RoboDK station: PDE4431_CW2_Final_Station4.rdk

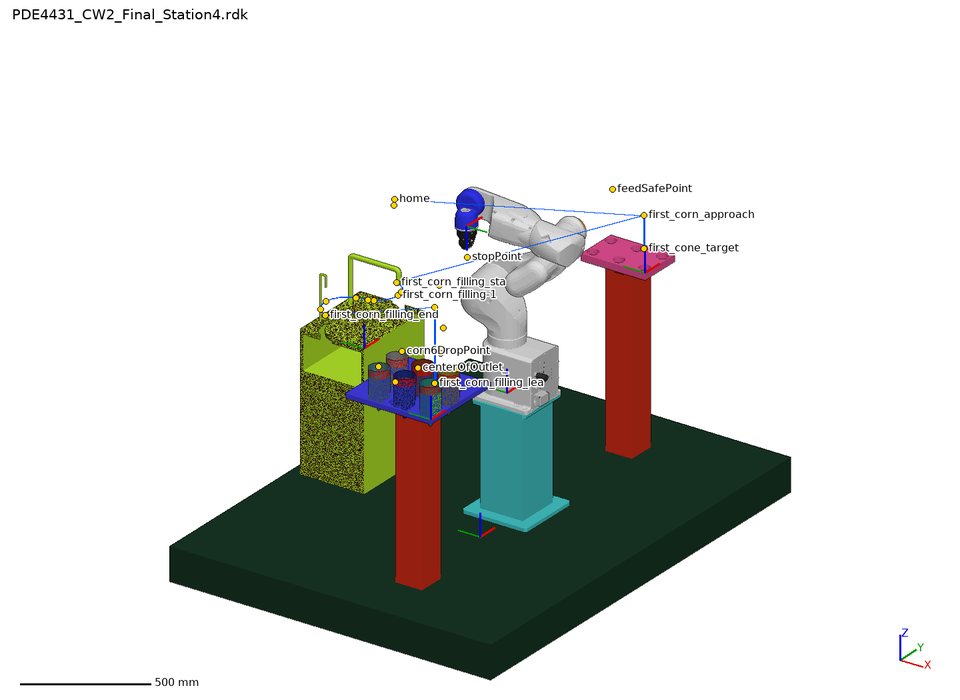
[picture v0: the station drawn from its stored meshes, robots at their saved joint values, targets as dots, program paths as lines]
Station PDE4431_CW2_Final_Station4 (saved by RoboDK 5.8.0). Poses are relative to the parent item; angles as X-Y-Z fixed-axis rotations.
  - frame world_frame at (0, 0, 10) mm, rotated rx 0 ry 0 rz 90 deg
    - object PDE4431_CW2_2024 at (0, 0, 0) mm, rotated rx 90 ry 0 rz 0 deg, size 2000 x 980 x 1500 mm, geometry from PDE4431_CW2_2024.STEP
    - object Pedestal_3 at (28, -150, 150) mm, rotated rx 90 ry 0 rz 0 deg, size 300 x 480 x 300 mm, geometry from Pedestal_3.STEP
    - frame Epson VT6 Base at (30, -105, 630) mm
      - robot Epson VT6: 6 axes, payload 6 kg, reach 920 mm, repeatability 0.1 mm, weight 40 kg
          modified DH rows (alpha deg, a mm, theta deg, d mm): 0, 0, 0, 412; -90, 100, -90, 0; 0, 420, 0, 0; -90, 0, 0, 400; 90, 0, 0, 0; -90, 0, 0, 80
          base shift (0, 0, 0) mm, rotated rx 0 ry 0 rz 90 deg
          joint limits [-170, -160, -51, -200, -125, -360] to [170, 65, 190, 200, 125, 360]; home [0, 0, 0, 0, 0, 0]; saved at [8.367, 49.246, -40.116, -0.033, -101.34, -10.833]
        - frame RobotiQ 2F-85 Gripper (Mechanism) Base at (0, 0, 0) mm, rotated rx 0 ry 0 rz 90 deg
          - robot RobotiQ 2F-85 Gripper (Mechanism) (model RobotiQ 2F85): 1 axes, payload 5 kg
              joint limits [0] to [85]; home [85]; saved at [60]
        - tool Tool 1, TCP at (0, 0, 130) mm
      - target gripper_open (Cartesian target) at (0, 683.92, 832) mm, rotated rx -90 ry 0 rz 0 deg; joints [85, 0, 0, 0, 0, 0] of RobotiQ 2F-85 Gripper (Mechanism)
      - target gripper_close (Cartesian target) at (0, 683.92, 832) mm, rotated rx -90 ry 0 rz 0 deg; joints [60, 0, 0, 0, 0, 0] of RobotiQ 2F-85 Gripper (Mechanism)
    - frame feed_frame at (600, -350, 980) mm
      - target home (Cartesian target) at (-608.8, 742.44, 350) mm, rotated rx 19.99 ry -88.06 rz -110.51 deg; joints [1.443, 8.858, -28.234, -5.378, 21.283, 5.738] of Epson VT6
      - target first_cone_target (Cartesian target) at (40.44, 31.41, 80) mm, rotated rx 9.95 ry -88.07 rz 169.53 deg; joints [-105.167, -26.118, -40.115, 15.72, 68.941, -5.939] of Epson VT6
      - target first_corn_approach (Cartesian target) at (40.44, 31.41, 220) mm, rotated rx 9.95 ry -88.07 rz 169.53 deg; joints [-123.826, -9.454, -31.705, 43.687, 52.628, -31.019] of Epson VT6
      - target first_corn_filling-1 (Cartesian target) at (-501.04, 802, -119.95) mm, rotated rx 9.87 ry -88.07 rz -104.39 deg; joints [-10.546, -59.86, -31.979, 6.038, 93.729, 0.524] of Epson VT6
      - target first_corn_filling_middle (Cartesian target) at (-598.8, 872.44, -119.95) mm, rotated rx 16 ry -88.06 rz -107 deg; joints [0.272, -60.26, -22.861, -1.267, 84.985, 0.686] of Epson VT6
      - target first_corn_filling-2 (Cartesian target) at (-698.8, 1000, -119.95) mm, rotated rx 9.99 ry -88.06 rz -100.51 deg; joints [8.938, -65.388, -0.069, -10.216, 67.714, 4.563] of Epson VT6
      - target first_corn_filling_end (Cartesian target) at (-798.8, 932.44, -119.95) mm, rotated rx 16 ry -88.06 rz -107 deg; joints [19.47, -63.29, -7.421, -21.334, 73.82, 7.44] of Epson VT6
      - target first_corn_filling_leave_point (Cartesian target) at (-1375, 18, 74.97) mm, rotated rx 30.01 ry -88.07 rz -30.53 deg; joints [103.327, -36.989, -18.254, -16.365, 58.039, 10.213] of Epson VT6
      - target first_corn_filling_retract_point (Cartesian target) at (-1375, 18, 400) mm, rotated rx 30.01 ry -88.07 rz -30.53 deg; joints [103.327, -12.172, 0.827, -47.435, 18.939, 47.222] of Epson VT6
      - target Target 11 (Cartesian target) at (-1337.42, 3.34, 300.08) mm, rotated rx 39.89 ry -88.07 rz -30.41 deg; joints [101.8, -15.291, -10.13, -5.083, 26.998, 5.831] of Epson VT6
      - target filling_cone_station1Mid (Cartesian target) at (-590, 852, -119.95) mm, rotated rx 9.87 ry -88.07 rz -104.39 deg; joints [0.759, -59.995, -25.833, -5.278, 87.745, 0.714] of Epson VT6
      - target filling_cone_middleMid (Cartesian target) at (-608.8, 922.44, -119.95) mm, rotated rx 9.99 ry -88.06 rz -110.51 deg; joints [4.755, -61.742, -14.063, -15.596, 78.219, 4.118] of Epson VT6
      - target filling_cone_station2Mid (Cartesian target) at (-768.8, 975, -119.95) mm, rotated rx 9.99 ry -88.06 rz -110.51 deg; joints [18.508, -65.639, 0.754, -31.046, 70.074, 12.988] of Epson VT6
      - target centerOfOutlet_ (Cartesian target) at (-1301, 148, 74.97) mm, rotated rx 30.01 ry -88.07 rz -30.53 deg; joints [90.451, -30.034, -33.078, -1.06, 64.789, 1.446] of Epson VT6
      - target corn2DropPoint (Cartesian target) at (-1451, 148, 74.97) mm, rotated rx 30.01 ry -88.07 rz -30.53 deg; joints [90.345, -42.143, -7.448, -1.095, 51.268, 1.676] of Epson VT6
      - target corn3DropPoint (Cartesian target) at (-1377, 278, 74.97) mm, rotated rx 30.01 ry -88.07 rz -30.53 deg; joints [77.46, -37.007, -18.216, 14.262, 57.748, -7.115] of Epson VT6
      - target corn4DropPoint (Cartesian target) at (-1225, 18, 79) mm, rotated rx 30.01 ry -88.07 rz -30.53 deg; joints [107.874, -25.434, -41.647, -19.605, 69.969, 8.477] of Epson VT6
      - target corn6DropPoint (Cartesian target) at (-1225, 278, 78) mm, rotated rx 30.01 ry -88.07 rz -30.53 deg; joints [73.098, -25.439, -42.006, 17.463, 70.07, -5.646] of Epson VT6
      - target corn5DropPoint (Cartesian target) at (-1151, 148, 78) mm, rotated rx 30.01 ry -88.07 rz -30.53 deg; joints [90.581, -19.834, -49.891, -1.149, 71.4, 1.364] of Epson VT6
      - target stopPoint (Cartesian target) at (-594.66, 411.86, 189.81) mm, rotated rx 179.62 ry 2.18 rz 87.53 deg; joints [7.54, 32.79, -35, 0, -90, -10] of Epson VT6
      - target feedSafePoint (Cartesian target) at (12.6, 160.61, 307.95) mm, rotated rx -176.96 ry -82.74 rz -13.55 deg; joints [-103.633, 8.826, -29.705, 13.041, 13.961, -12.658] of Epson VT6
      - target fillingSafePoint (Cartesian target) at (-581.1, 764.07, 307.97) mm, rotated rx 13.01 ry -87.26 rz -103.52 deg; joints [-1.569, 31.922, -49.422, 3.122, 20.195, -2.364] of Epson VT6
      - target outletSafePoint (Cartesian target) at (-1053.51, 222.32, 307.96) mm, rotated rx 0 ry -90 rz -0.51 deg; joints [95.528, 33.432, -48.583, -22.02, 16.282, 21.217] of Epson VT6
      - target first_corn_filling_start (Cartesian target) at (-408.8, 872.44, -119.95) mm, rotated rx 16 ry -88.06 rz -110.51 deg; joints [-24.103, -60.578, -38.406, 19.925, 100.319, 3.586] of Epson VT6
      - target filling_cone_startMid (Cartesian target) at (-468.8, 808, -119.95) mm, rotated rx 16 ry -88.06 rz -110.51 deg; joints [-19.022, -64.883, -48.536, 15.982, 114.48, 6.82] of Epson VT6
      - target Target 27 (Cartesian target) at (-590, 852, -119.95) mm, rotated rx 9.87 ry -88.07 rz -104.39 deg; joints [2.722, -62.994, -45.373, -7.708, 110.114, -2.093] of Epson VT6
    - frame outlet_frame at (-900, -400, 970) mm
      - object Corn1 at (40, 30, 50) mm, rotated rx 90 ry 0.08 rz 0 deg, size 84.9 x 182 x 85 mm, geometry from Cone-Part.STEP
      - object Corn2 at (40, 150, 50) mm, rotated rx 90 ry 0 rz 0 deg, size 84.9 x 182 x 85 mm, geometry from Cone-Part.STEP
      - object Corn3 at (40, 270, 50) mm, rotated rx 90 ry 0 rz 0 deg, size 84.9 x 182 x 85 mm, geometry from Cone-Part.STEP
      - object Corn4 at (160, 30, 50) mm, rotated rx 90 ry 0 rz 0 deg, size 84.9 x 182 x 85 mm, geometry from Cone-Part.STEP
      - object Corn5 at (160, 150, 50) mm, rotated rx 90 ry 0 rz 0 deg, size 84.9 x 182 x 85 mm, geometry from Cone-Part.STEP
      - object Corn6 at (160, 270, 50) mm, rotated rx 90 ry 0 rz 0 deg, size 84.9 x 182 x 85 mm, geometry from Cone-Part.STEP
    - frame filling_station_frame at (-200, 400, 770) mm
  - program gripper_open (2 instructions, listed below)
  - program gripper_close (2 instructions, listed below)
  - program mainProgram (20 instructions, listed below)
  - program Replace_Corns (1 instructions, listed below)
  - Python program firstCornProgramInPython (listed below)
  - program AttachObject1 (1 instructions, listed below)
  - program DeattachObject1 (1 instructions, listed below)
  - Python program mainAllCornProgramInPython (listed below)
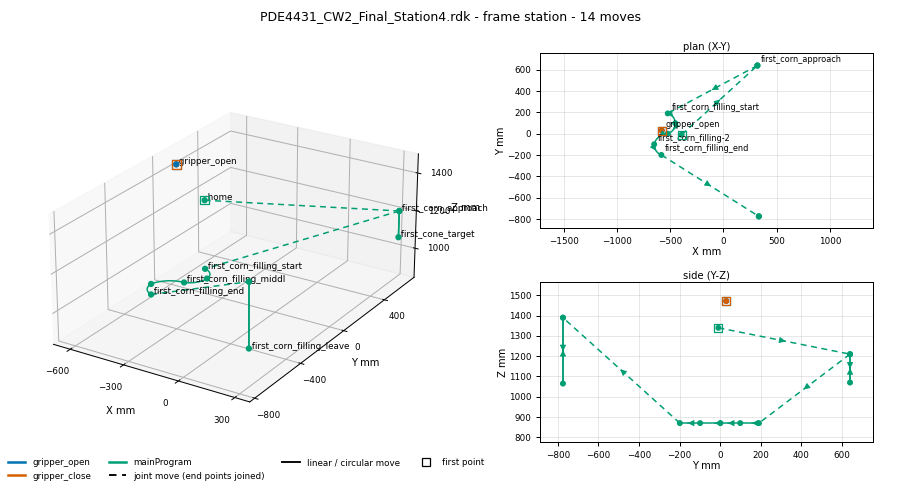
[picture p0: tool path of PDE4431_CW2_Final_Station4.rdk in frame station, 14 of 14 moves have a stored position in this frame; points joined in program order, loops and branches not executed]

--- program gripper_open (robot RobotiQ 2F-85 Gripper (Mechanism)) ---
  Set Ref.: Epson VT6 Base
  MoveJ (gripper_open)

--- program gripper_close (robot RobotiQ 2F-85 Gripper (Mechanism)) ---
  Set Ref.: Epson VT6 Base
  MoveJ (gripper_close)

--- program mainProgram (robot Epson VT6) ---
  MoveJ (home)
  MoveJ (first_corn_approach)
  Call gripper_open
  Set Ref.: feed_frame
  Set Tool: Tool 1
  MoveL (first_cone_target)
  Call gripper_close
  Attach to Tool 1
  MoveL (first_corn_approach)
  MoveJ (first_corn_filling_start)
  MoveC (filling_cone_startMid, first_corn_filling-1)
  MoveC (filling_cone_station1Mid, first_corn_filling_middle)
  MoveC (filling_cone_middleMid, first_corn_filling-2)
  MoveC (filling_cone_station2Mid, first_corn_filling_end)
  MoveJ (first_corn_filling_retract_point)
  MoveL (first_corn_filling_leave_point)
  Call gripper_open
  Detach from Tool 1
  MoveL (first_corn_filling_retract_point)
  Set speed (500.0 mm/s)

--- program Replace_Corns (robot Epson VT6) ---
  Replace objects

--- Python program firstCornProgramInPython ---
from robodk.robolink import *  # Import the RoboDK API
from robodk.robomath import *  # Import RoboDK math utilities
import time

# Establishing the connection with RoboDK Robot
RDK = Robolink()  # Correctly instantiate the RoboDK connection

# Configuring two different robots as RoboDK items
robot_1 = RDK.Item('Epson VT6')  # Select the robot by name
feed_frame = RDK.Item('feed_frame')    # Initial frame of the object
outlet_frame = RDK.Item('outlet_frame')# Final frame for the object


if not robot_1.Valid():
    print("Error: Robot not found or invalid item")
    quit()

# Select the home target
homeNew = RDK.Item('home')
#Feed frame Section
first_corn_approach = RDK.Item('first_corn_approach')
first_corn_target = RDK.Item('first_cone_target')

#Filling frame Section
filling_start = RDK.Item('first_corn_filling_start')
filling_cone_startMid = RDK.Item('filling_cone_startMid')
filling_station_1 = RDK.Item('first_corn_filling-1')
filling_cone_station1Mid = RDK.Item('filling_cone_station1Mid')
filling_middle = RDK.Item('first_corn_filling_middle')
filling_cone_middleMid = RDK.Item('filling_cone_middleMid')
filling_station_2 = RDK.Item('first_corn_filling-2')
filling_cone_station2Mid = RDK.Item('filling_cone_station2Mid')
filling_end = RDK.Item('first_corn_filling_end')

#Outlet frame Section
first_corn_filling_retract_point = RDK.Item('first_corn_filling_retract_point')
first_corn_filling_leave_point = RDK.Item('first_corn_filling_leave_point')

# Run a Python script program
gripper_open = RDK.Item('gripper_open', ITEM_TYPE_PROGRAM)  # For gripper open
gripper_close = RDK.Item('gripper_close', ITEM_TYPE_PROGRAM)  # For gripper close


# Find the object to attach
object_to_attach = RDK.Item('Corn1')  # Replace 'Cone' with the name of your object

# Attach the object to the robot's tool
tool = robot_1.Childs()[0]  # Get the robot's tool (or specify the tool name directly)

if object_to_attach.Valid() and tool.Valid():
    print("Object and Tool set successfully.")
else:
    print("Error: Object and/or Tool is not valid.")

def TCP_On():
    current_pose = object_to_attach.PoseAbs()
    object_to_attach.setParent(tool)
    object_to_attach.setPoseAbs(current_pose)
    print("Object attached to the tool.")

def TCP_Off():

    current_pose = object_to_attach.PoseAbs()
    object_to_attach.setParent(outlet_frame)
    object_to_attach.setPoseAbs(current_pose)
    print("Object detached from the tool and reattached to Outlet Frame.")


# Set the speed of the robot
robot_1.setSpeed(50)  # Use the method on the robot item

robot_1.MoveJ(homeNew)
robot_1.MoveJ(first_corn_approach)
gripper_open.RunCode()
time.sleep(0.5)
robot_1.MoveL(first_corn_target)
gripper_close.RunCode()
TCP_On()
time.sleep(0.5)
robot_1.MoveL(first_corn_approach)
robot_1.MoveJ(filling_start)
robot_1.MoveC(filling_cone_startMid, filling_station_1)
time.sleep(1)
robot_1.MoveC(filling_cone_station1Mid, filling_middle)
robot_1.MoveC(filling_cone_middleMid, filling_station_2)
time.sleep(1)
robot_1.MoveC(filling_cone_station2Mid, filling_end)
robot_1.MoveJ(first_corn_filling_retract_point)
robot_1.MoveL(first_corn_filling_leave_point)
gripper_open.RunCode()
time.sleep(0.5)
TCP_Off()
time.sleep(0.5)
robot_1.MoveL(first_corn_filling_retract_point)
robot_1.MoveJ(homeNew)

--- program AttachObject1 (robot Epson VT6) ---
  Attach to Tool 1

--- program DeattachObject1 (robot Epson VT6) ---
  Detach from Tool 1

--- Python program mainAllCornProgramInPython ---
from robodk.robolink import *  # Import the RoboDK API
from robodk.robomath import transl, rotz
from math import radians, cos, sin, atan2  # Use the standard math module
import time
import math

# Establishing the connection with RoboDK Robot
RDK = Robolink()  # Correctly instantiate the RoboDK connection

# Configuring two different robots as RoboDK items
robot_1 = RDK.Item('Epson VT6')  # Select the robot by name
feed_frame = RDK.Item('feed_frame')    # Initial frame of the object
outlet_frame = RDK.Item('outlet_frame')# Final frame for the object


if not robot_1.Valid():
    print("Error: Robot not found or invalid item")
    quit()

# Select the home target
homeNew = RDK.Item('home')
#Feed frame Section
first_corn_approach = RDK.Item('first_corn_approach')
first_corn_target = RDK.Item('first_cone_target')

cone1App_pos = RDK.Item("first_corn_approach")
secondApp_target =  cone1App_pos.Pose()*transl(0, -120, 0)
thirdApp_target =  cone1App_pos.Pose()*transl(0, -240, 0)
forthApp_target =  cone1App_pos.Pose()*transl(0, 0, 120)
fifthApp_target =  cone1App_pos.Pose()*transl(0, -120, 120)
sixthApp_target =  cone1App_pos.Pose()*transl(0, -240, 120)

approachPoints = [first_corn_approach, secondApp_target, thirdApp_target, forthApp_target, fifthApp_target, sixthApp_target]

cone1_pos = RDK.Item("first_cone_target")
second_target =  cone1_pos.Pose()*transl(0, -120, 0)
third_target =  cone1_pos.Pose()*transl(0, -240, 0)
forth_target =  cone1_pos.Pose()*transl(0, 0, 120)
fifth_target =  cone1_pos.Pose()*transl(0, -120, 120)
sixth_target =  cone1_pos.Pose()*transl(0, -240, 120)

targetPoints = [first_corn_target, second_target, third_target, forth_target, fifth_target, sixth_target]

cone_names = [
    'Corn1','Corn2','Corn3','Corn4','Corn5','Corn6',
]

#Filling frame Section
filling_start = RDK.Item('first_corn_filling_start')
filling_cone_startMid = RDK.Item('filling_cone_startMid')
filling_station_1 = RDK.Item('first_corn_filling-1')
filling_cone_station1Mid = RDK.Item('filling_cone_station1Mid')
filling_middle = RDK.Item('first_corn_filling_middle')
filling_cone_middleMid = RDK.Item('filling_cone_middleMid')
filling_station_2 = RDK.Item('first_corn_filling-2')
filling_cone_station2Mid = RDK.Item('filling_cone_station2Mid')
filling_end = RDK.Item('first_corn_filling_end')

feedSafePoint = RDK.Item('feedSafePoint')
fillingSafePoint = RDK.Item('fillingSafePoint')
outletSafePoint = RDK.Item('outletSafePoint')

hexagonCenter = RDK.Item('centerOfOutlet_')  #hexagon center

#Outlet frame Section
first_corn_filling_retract_point = RDK.Item('first_corn_filling_leave_point').Pose()*transl(150.00, 0, 0)
corn2_RetractPoint = RDK.Item("corn2DropPoint").Pose()*transl(150.00, 0, 0)
corn3_RetractPoint = RDK.Item("corn3DropPoint").Pose()*transl(150.00, 0, 0)
corn4_RetractPoint = RDK.Item("corn4DropPoint").Pose()*transl(150.00, 0, 0)
corn5_RetractPoint = RDK.Item("corn5DropPoint").Pose()*transl(150.00, 0, 0)
corn6_RetractPoint = RDK.Item("corn6DropPoint").Pose()*transl(150.00, 0, 0)

first_corn_filling_leave_point = RDK.Item('first_corn_filling_leave_point')
corn2DropPoint = RDK.Item('corn2DropPoint')
corn3DropPoint = RDK.Item('corn3DropPoint')
corn4DropPoint = RDK.Item('corn4DropPoint')
corn5DropPoint = RDK.Item('corn5DropPoint')
corn6DropPoint = RDK.Item('corn6DropPoint')

stopPoint = RDK.Item('stopPoint')

outlet_retractPoint = [first_corn_filling_retract_point, corn2_RetractPoint, corn3_RetractPoint, corn4_RetractPoint, corn5_RetractPoint, corn6_RetractPoint]
outlet_targetPoint = [first_corn_filling_leave_point, corn2DropPoint, corn3DropPoint, corn4DropPoint, corn5DropPoint, corn6DropPoint]


# Run a Python script program
gripper_open = RDK.Item('gripper_open', ITEM_TYPE_PROGRAM)  # For gripper open
gripper_close = RDK.Item('gripper_close', ITEM_TYPE_PROGRAM)  # For gripper close
Replace_Corns = RDK.Item('Replace_Corns', ITEM_TYPE_PROGRAM)  # For Cones back to feed frame


# Find the object to attach
object_to_attach = RDK.Item('Corn1')  # Replace 'Cone' with the name of your object

# Attach the object to the robot's tool
tool = robot_1.Childs()[0]  # Get the robot's tool (or specify the tool name directly)

if object_to_attach.Valid() and tool.Valid():
    print("Object and Tool set successfully.")
else:
    print("Error: Object and/or Tool is not valid.")

def TCP_On(object_to_attach):
    object_to_attach = RDK.Item(object_to_attach)
    current_pose = object_to_attach.PoseAbs()
    object_to_attach.setParent(tool)
    object_to_attach.setPoseAbs(current_pose)
    print("Object attached to the tool.")

def TCP_Off(object_to_attach):
    object_to_attach = RDK.Item(object_to_attach)
    current_pose = object_to_attach.PoseAbs()
    object_to_attach.setParent(outlet_frame)
    object_to_attach.setPoseAbs(current_pose)
    print("Object detached from the tool and reattached to Outlet Frame.")

def main():
    robot_1.setSpeed(100)  # Use the method on the robot item
    Replace_Corns.RunCode()
    robot_1.MoveJ(homeNew)

    for n in range(6):
        robot_1.MoveJ(feedSafePoint)
        robot_1.MoveJ(approachPoints[n])
        gripper_open.RunCode()
        time.sleep(0.5)
        robot_1.MoveL(targetPoints[n])
        gripper_close.RunCode()
        time.sleep(1)
        TCP_On(cone_names[n])
        time.sleep(1)
        robot_1.MoveL(approachPoints[n])
        robot_1.MoveJ(feedSafePoint)
        robot_1.MoveJ(fillingSafePoint)
        filling_retractPoint = filling_start.Pose()*transl(150.00, 0, 0)
        robot_1.MoveJ(filling_retractPoint)
        robot_1.MoveJ(filling_start)

        robot_1.MoveC(filling_cone_startMid, filling_station_1)
        # robot_1.MoveJ(filling_cone_startMid)
        # robot_1.MoveJ(filling_station_1)

        time.sleep(1)

        robot_1.MoveC(filling_cone_station1Mid, filling_middle)
        # robot_1.MoveJ(filling_cone_station1Mid)
        # robot_1.MoveJ(filling_middle)

        robot_1.MoveC(filling_cone_middleMid, filling_station_2)
        # robot_1.MoveJ(filling_cone_middleMid)
        # robot_1.MoveJ(filling_station_2)

        time.sleep(1)

        # robot_1.MoveC(filling_cone_station2Mid, filling_end)
        robot_1.MoveJ(filling_cone_station2Mid)
        robot_1.MoveJ(filling_end)

        fillingEnd_retractPoint = filling_end.Pose()*transl(150.00, 0, 0)
        robot_1.MoveJ(fillingEnd_retractPoint)
        robot_1.MoveJ(fillingSafePoint)
        robot_1.MoveJ(outletSafePoint)
        robot_1.MoveJ(outlet_retractPoint[n])
        robot_1.MoveL(outlet_targetPoint[n])
        gripper_open.RunCode()
        time.sleep(0.5)
        TCP_Off(cone_names[n])
        time.sleep(0.5)
        robot_1.MoveL(outlet_retractPoint[n])
        robot_1.MoveJ(outletSafePoint)

    robot_1.MoveJ(stopPoint)

main()
